TYPE EnableRtsCts EXTENDS SubIndexModuleBase :
STRUCT
END_STRUCT
END_TYPE

(* stored: Version 1.1.0.1, ProductVersion 3.1.4024.3
   DUT EnableRtsCts: Id {8b7125bf-7b5c-46d9-a9bf-780d6aeedf4d} *)
